// TIA Portal project "es003_nastro_con_timer" (V16)

(* hardware
DEVICE "S7-1200 station_1"  S7-1200 Station
   slot 0: "Telaio di montaggio_0"  S7-1200 Rack  Rack  V1.0
   slot 1: "PLC_1"  CPU 1215C DC/DC/Rly  6ES7 215-1HG40-0XB0  V4.2
*)

// ===== PLC "PLC_1"  CPU 1215C DC/DC/Rly =====

DATA_BLOCK "Dati_HMI"   // DB1
{ S7_Optimized_Access := 'TRUE' }
VERSION : 0.1
   VAR
      jog_start : Bool;
      jog_ripristino : Bool;
      jog_bc_inizio : Bool;
      jog_bc_fine : Bool;
      avanti_nastro : Bool;
      indietro_nastro : Bool;
      passo_0 : Bool;
      passo_1 : Bool;
      passo_2 : Bool;
      passo_3 : Bool;
      t_delay : Bool;
      mem_preset : Time;
      caricamento_preset : Bool;
      inserisci_tempo : Time;
      conteggio_corrente : Time;
   END_VAR
BEGIN
END_DATA_BLOCK

// folder: System blocks/Program resources

DATA_BLOCK "Timer_attesa_lavorazione"   // DB2
{ S7_Optimized_Access := 'TRUE' }
AUTHOR : Simatic
FAMILY : IEC
NAME : IEC_TMR
VERSION : 1.0
// stored: InstanceOfName IEC_TIMER
"IEC_TIMER"
BEGIN
END_DATA_BLOCK

// folder: (top level)

FUNCTION "Ripristino" : Void   // FC1, LAD
{ S7_Optimized_Access := 'TRUE' }
VERSION : 0.1
BEGIN

REGION Network 1
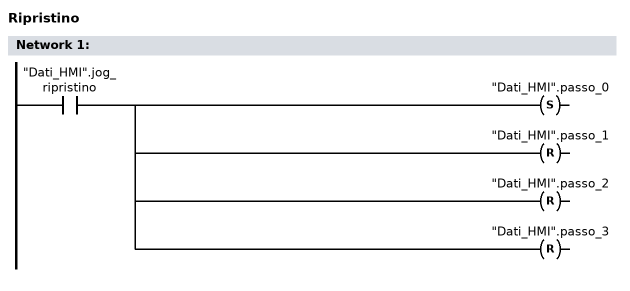
   RUNG wire#powerrail
      Contact( "Dati_HMI".jog_ripristino )
      wire#w1
      S_Coil( "Dati_HMI".passo_0 )
   END_RUNG
   RUNG wire#w1
      R_Coil( "Dati_HMI".passo_1 )
   END_RUNG
   RUNG wire#w1
      R_Coil( "Dati_HMI".passo_2 )
   END_RUNG
   RUNG wire#w1
      R_Coil( "Dati_HMI".passo_3 )
   END_RUNG
   // the same network as SCL:
   IF "Dati_HMI".jog_ripristino THEN
       "Dati_HMI".passo_0 := TRUE;
       "Dati_HMI".passo_1 := FALSE;
       "Dati_HMI".passo_2 := FALSE;
       "Dati_HMI".passo_3 := FALSE;
   END_IF;
END_REGION
END_FUNCTION

FUNCTION "Struttura_passi" : Void   // FC2, LAD
{ S7_Optimized_Access := 'TRUE' }
VERSION : 0.1
BEGIN

REGION Network 1
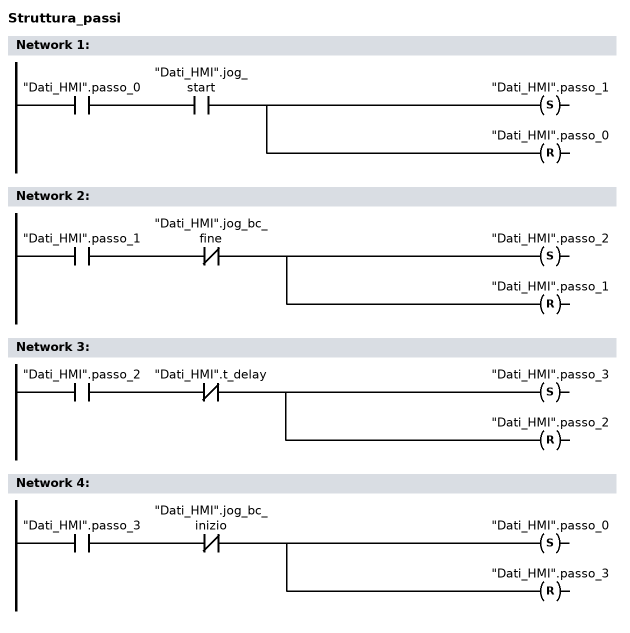
   RUNG wire#powerrail
      Contact( "Dati_HMI".passo_0 )
      Contact( "Dati_HMI".jog_start )
      wire#w1
      S_Coil( "Dati_HMI".passo_1 )
   END_RUNG
   RUNG wire#w1
      R_Coil( "Dati_HMI".passo_0 )
   END_RUNG
   // the same network as SCL:
   IF "Dati_HMI".passo_0 AND "Dati_HMI".jog_start THEN
       "Dati_HMI".passo_1 := TRUE;
       "Dati_HMI".passo_0 := FALSE;
   END_IF;
END_REGION

REGION Network 2
   RUNG wire#powerrail
      Contact( "Dati_HMI".passo_1 )
      I_Contact( "Dati_HMI".jog_bc_fine )
      wire#w1
      S_Coil( "Dati_HMI".passo_2 )
   END_RUNG
   RUNG wire#w1
      R_Coil( "Dati_HMI".passo_1 )
   END_RUNG
   // the same network as SCL:
   IF "Dati_HMI".passo_1 AND NOT "Dati_HMI".jog_bc_fine THEN
       "Dati_HMI".passo_2 := TRUE;
       "Dati_HMI".passo_1 := FALSE;
   END_IF;
END_REGION

REGION Network 3
   RUNG wire#powerrail
      Contact( "Dati_HMI".passo_2 )
      I_Contact( "Dati_HMI".t_delay )
      wire#w1
      S_Coil( "Dati_HMI".passo_3 )
   END_RUNG
   RUNG wire#w1
      R_Coil( "Dati_HMI".passo_2 )
   END_RUNG
   // the same network as SCL:
   IF "Dati_HMI".passo_2 AND NOT "Dati_HMI".t_delay THEN
       "Dati_HMI".passo_3 := TRUE;
       "Dati_HMI".passo_2 := FALSE;
   END_IF;
END_REGION

REGION Network 4
   RUNG wire#powerrail
      Contact( "Dati_HMI".passo_3 )
      I_Contact( "Dati_HMI".jog_bc_inizio )
      wire#w1
      S_Coil( "Dati_HMI".passo_0 )
   END_RUNG
   RUNG wire#w1
      R_Coil( "Dati_HMI".passo_3 )
   END_RUNG
   // the same network as SCL:
   IF "Dati_HMI".passo_3 AND NOT "Dati_HMI".jog_bc_inizio THEN
       "Dati_HMI".passo_0 := TRUE;
       "Dati_HMI".passo_3 := FALSE;
   END_IF;
END_REGION
END_FUNCTION

FUNCTION "Attivazione_uscite" : Void   // FC3, LAD
{ S7_Optimized_Access := 'TRUE' }
VERSION : 0.1
BEGIN

REGION Network 1
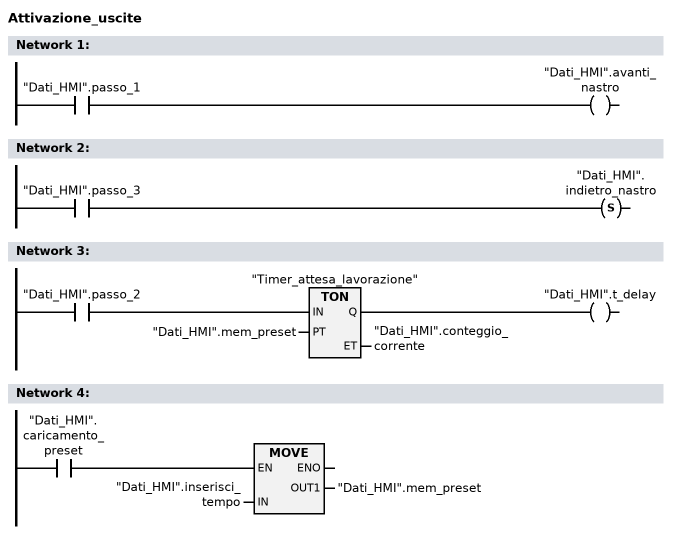
   RUNG wire#powerrail
      Contact( "Dati_HMI".passo_1 )
      Coil( "Dati_HMI".avanti_nastro )
   END_RUNG
   // the same network as SCL:
   "Dati_HMI".avanti_nastro := "Dati_HMI".passo_1;
END_REGION

REGION Network 2
   RUNG wire#powerrail
      Contact( "Dati_HMI".passo_3 )
      S_Coil( "Dati_HMI".indietro_nastro )
   END_RUNG
   // the same network as SCL:
   IF "Dati_HMI".passo_3 THEN "Dati_HMI".indietro_nastro := TRUE; END_IF;
END_REGION

REGION Network 3
   "Timer_attesa_lavorazione".TON(IN := "Dati_HMI".passo_2,
                           PT := "Dati_HMI".mem_preset,
                           ET => "Dati_HMI".conteggio_corrente);
   "Dati_HMI".t_delay := "Timer_attesa_lavorazione".Q;
END_REGION

REGION Network 4
   RUNG wire#powerrail
      Contact( "Dati_HMI".caricamento_preset )
      Move(in := "Dati_HMI".inserisci_tempo, out1 => "Dati_HMI".mem_preset)
   END_RUNG
   // the same network as SCL:
   IF "Dati_HMI".caricamento_preset THEN "Dati_HMI".mem_preset := "Dati_HMI".inserisci_tempo; END_IF;
END_REGION
END_FUNCTION

ORGANIZATION_BLOCK "Main"   // OB1, LAD, ProgramCycle
TITLE = "Main Program Sweep (Cycle)"
{ S7_Optimized_Access := 'TRUE' }
VERSION : 0.1
   VAR_INPUT
      Initial_Call : Bool;   // Initial call of this OB
      Remanence : Bool;   // =True, if remanent data are available
   END_VAR
BEGIN

REGION Network 1
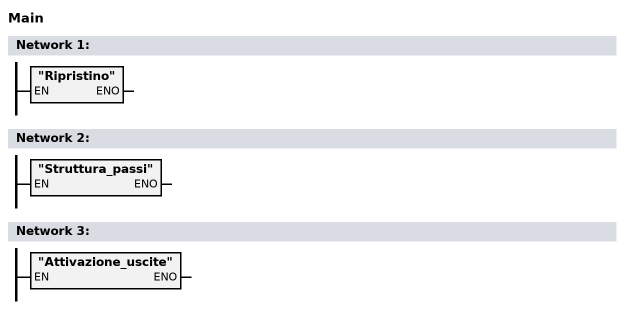
   RUNG wire#powerrail
      "Ripristino"()
   END_RUNG
   // the same network as SCL:
   "Ripristino"();
END_REGION

REGION Network 2
   RUNG wire#powerrail
      "Struttura_passi"()
   END_RUNG
   // the same network as SCL:
   "Struttura_passi"();
END_REGION

REGION Network 3
   RUNG wire#powerrail
      "Attivazione_uscite"()
   END_RUNG
   // the same network as SCL:
   "Attivazione_uscite"();
END_REGION
END_ORGANIZATION_BLOCK